FUNCTION_BLOCK FB_PfeifferTurboPump EXTENDS FB_TurboPump
VAR_INPUT
END_VAR
VAR_OUTPUT
END_VAR
VAR
END_VAR

SUPER^.PumpLogic();

END_FUNCTION_BLOCK

(* stored: Version 1.1.0.1, ProductVersion 3.1.4020.12
   POU FB_PfeifferTurboPump: Id {8a094e05-8b3e-4241-abfb-693b3ec2b80c}, SpecialFunc None *)
